FUNCTION_BLOCK PlixHandler
VAR_INPUT
	go :BOOL;

END_VAR
VAR_OUTPUT
	

END_VAR
VAR
	//Arduino				/////////////////////////////////////////
		//States
	Scanner					:USINT		:= 10;
	
		//Varibles
	WingUp					:USINT 		:=220;
	WingFlat				:USINT 		:=180;
	WingHDown				:USINT 		:=155;
	WingDown				:USINT 		:=80;
	WiggleDown				:USINT 		:=155;
	WiggleUP				:USINT 		:=190;
	FanHigh					:USINT 		:=115;
	FanLow					:USINT 		:=95;
	FanOff					:USINT 		:=89;
	FanReverse				:USINT 		:=74;
	WingGo					:USINT		:=20;
	FanGo					:USINT		:=30;

	//Stepper				/////////////////////////////////////////
	HaltStackStepper	: MC_Halt;
	EnableStackStepper	: MC_Power;
	MoveStackAbsolute	: MC_MoveAbsolute;
	ReadStackPosition	: MC_ReadActualPosition;
	SetStackPosition	: MC_SetPosition;
	StopStackStepper	: MC_Stop;
	ResetStackStepper	: MC_Reset;
	
		//Varibles
	StackStepperRun: BOOL;
	StackStepperPosition: LREAL;
	StackStepperVelocity: LREAL;
	StackStepperCurrentPosition: LREAL;
	StackStepperZeroPosition : BOOL;
	StackStepperStop: BOOL;
	StackStepperReset: BOOL;
	StackStepperHalt: BOOL;
	StackStepperHaltDone: BOOL;
	StackStepperAbsoluteDone: BOOL;
	StackStepperEnable: BOOL;
	
	Byte31IN: BYTE;
	StackSensor1: BOOL;
	Sensors: BYTE;
	StackSensor2: BOOL;
	StackSensor3: BOOL;
	Sensor4: BOOL;
	Sensor5: BOOL;
	PlixHandlerState: INT;
	BottomEndStop: BOOL;
	Boot: BOOL := TRUE;
	Calibrate 				:BOOL;
	NextState: INT;
	Single					:BOOL;
	Double					:BOOL;
	Zero					:BOOL;
	Start					:BOOL;
	//Stats					/////////////////////////////////////////
	Singles					:INT;
	Doubles					:INT;
	Zeros					:INT;
	Total					:INT;
	Wiggle					:INT;
	Count 					:INT		:= 0;
	Delay 					:TON;
	CycleTime				:REAL;
	EndTime					:REAL;
	AverageTime				:REAL;
	DoubleLoop: INT;
	Blast: BOOL;
	Cali: INT	 :=0;
	Velocity 				:LREAL :=800;
	ErrorID1		        : UDINT;
	
	Pig: BOOL;
END_VAR
VAR PERSISTENT				/////////////////////////////////////////
	
	//CutPoints				/////////////////////////////////////////
	PlixNumberScan			:INT;
	PlixNumberScanLeft		:INT;
	PlixNumberScanRight		:INT;
	NormalTopCut			:UINT;
	NormalBottomCut			:UINT;
	TopCut					:UINT;
	BottomCut				:UINT;
	DoubleTopCut			:UINT;
	DoubleBottomCut			:UINT;
	TopCutLeft				:INT;
	BottomCutLeft			:INT;
	TopCutRight				:INT;
	BottomCutRight			:INT;
	
	
	//Time					/////////////////////////////////////////

END_VAR

MoveStackAbsolute(
	Axis:= GVL.StackStepper, 
	Execute:= StackStepperRun, 
	Position:= StackStepperPosition, 
	Velocity:= StackStepperVelocity, 
	Acceleration:= 2518.53, 
	Deceleration:= 2518.53, 
	Jerk:= 10703.7,
	Done=> StackStepperAbsoluteDone, );
	
HaltStackStepper(
	Axis:= GVL.StackStepper, 
	Execute:= StackStepperHalt, 
	Deceleration:= 2518.53,  
	Done=> StackStepperHaltDone,
	ErrorID=> ErrorID1, );
	
EnableStackStepper(
	Axis:= GVL.StackStepper, 
	Enable:= StackStepperEnable, 
	Enable_Positive:= StackStepperEnable, 
	Enable_Negative:= StackStepperEnable, );

ReadStackPosition(
	Axis:= GVL.StackStepper, 
	Enable:= StackStepperEnable, 
	Position=> StackStepperCurrentPosition);	

SetStackPosition(
	Axis:= GVL.StackStepper, 
	Execute:= StackStepperZeroPosition, 
	Position:= 0, 
	Mode:= FALSE, 
	Options:= , 
	 );
	
StopStackStepper(
	Axis:= GVL.StackStepper, 
	Execute:= StackStepperStop, 
	Deceleration:= , 
	Jerk:= , 
	Options:= , 
	Done=> , 
	Busy=> , 
	Active=> , 
	CommandAborted=> , 
	Error=> , 
	ErrorID=> );
	
ResetStackStepper(
	Axis:= GVL.StackStepper, 
	Execute:= StackStepperReset, 
	Done=> , 
	Busy=> , 
	Error=> , 
	ErrorID=> );
	
	
	
	
	//Coms

IF go THEN
	StackStepperEnable := TRUE;
END_IF
StackSensor2 := GVL.Sensors2.0;
BottomEndStop :=GVL.Sensors2.1;
//StackStepperZeroPosition := TRUE;//sometimes after many restarts the position can be massive and cause problems 


CASE PlixHandlerState OF
	
	1:
		StackStepperZeroPosition := FALSE;
		StackStepperRun := FALSE;
		StackStepperHalt :=TRUE;
		IF StackStepperHaltDone THEN 
				PlixHandlerState :=NextState;
				StackStepperHalt :=FALSE;
		END_IF
		
	
	10:	
		IF Boot THEN
			StackStepperZeroPosition := TRUE;
			PlixHandlerState := 11;
		ELSE
			PlixHandlerState := 100;
		END_IF
		
	11://home bottom sensor
		StackStepperZeroPosition := FALSE;
		IF  BottomEndStop THEN//if not blocked drive down till blocked
			StackStepperPosition := -50000;
			StackStepperVelocity := 100;
			StackStepperRun := TRUE;
		ELSE 
			NextState :=20;
			PlixHandlerState :=1;
				
		END_IF
		
	20:
		IF  NOT BottomEndStop THEN//drive up till unblocked
			StackStepperPosition := 8000;
			StackStepperVelocity := 100;
			StackStepperRun := TRUE;
		ELSE 
			NextState :=30;
			PlixHandlerState :=1;	
		END_IF	
		
	30:
		Boot := FALSE;
		StackStepperZeroPosition := TRUE;//set position to zero just above endstop
		//StackStepperZeroPosition := FALSE;
		PlixHandlerState :=100;
	
	100:// home stack top
		StackStepperZeroPosition := FALSE;
		IF NOT StackSensor2 THEN//AND NOT StackSensor2 AND NOT StackSensor3 THEN
			StackStepperPosition := 200;
			StackStepperVelocity := Velocity;//make sure to change the amount of steps to plix pick up
			StackStepperRun := TRUE;
		ELSE 
			NextState :=200;
			PlixHandlerState :=1;
			
		END_IF
	200:
		StackStepperHalt :=FALSE;
		IF StackSensor2 THEN//AND  StackSensor2 AND  StackSensor3 THEN
			StackStepperPosition := 10000;
			StackStepperVelocity := Velocity;//make sure to change the amount of steps to plix pick up
			StackStepperRun := TRUE;
		ELSE 
			NextState :=300;
			PlixHandlerState :=1;
				
		END_IF
	300://fan on
		IF GVL.ArduinoBusyBit THEN//if  arduino is free then ask to change state
			GVL.FanDyno := FanHigh;
			GVL.ArduinoState := FanGo;
			PlixHandlerState :=400;
		END_IF
		
	400://up to head
		IF Blast THEN 
			GVL.StackBlast := TRUE;
		END_IF
		Blast := FALSE;
		StackStepperHalt :=FALSE;
		StackStepperPosition := StackStepperCurrentPosition + 50;
		StackStepperVelocity := Velocity;
		StackStepperRun := TRUE;
		PlixHandlerState :=500;
		
	500://down
		
		StackStepperRun := FALSE;
		IF StackStepperAbsoluteDone THEN
			GVL.StackBlast := FALSE;
		/////
			
			StackStepperPosition := StackStepperCurrentPosition - 400;
			StackStepperVelocity := Velocity;//make sure to change the amount of steps to plix pick up
			StackStepperRun := TRUE;
			StackStepperAbsoluteDone := FALSE;
			PlixHandlerState :=550;
			
		END_IF
		
	550:
		StackStepperRun := FALSE;
		IF StackStepperAbsoluteDone THEN
			NextState :=575;
			PlixHandlerState :=1;
				
		END_IF
		
	575:
		IF Calibrate THEN
			PlixHandlerState :=580;
		ELSE
			PlixHandlerState :=600;
		END_IF
		
	580:
		Delay(IN:=TRUE, PT:=T#1000MS);
      	IF Delay.Q THEN
        	Delay(IN:=FALSE);
			
			PlixHandlerState :=600;
		END_IF
	600://scan
		
		IF GVL.ArduinoBusyBit THEN//if arduino is free then ask to change state
			GVL.ArduinoState := Scanner;
			PlixHandlerState :=700;
		END_IF
	
	700:
		IF GVL.ArduinoBusyBit THEN//if arduino is free then ask to change state
			PlixHandlerState :=800;
		END_IF
	800://still hasnt written the new scan to beckhoff so we need to wait a little for it to loop on the arduino
	Delay(IN:=TRUE, PT:=T#500MS);
      	IF Delay.Q THEN
        	Delay(IN:=FALSE);
			
			PlixHandlerState :=900;
		END_IF
	900:
		IF NOT Calibrate THEN
			IF DoubleLoop > 0 THEN
				TopCut := DoubleTopCut;
				BottomCut := DoubleBottomCut;
				PlixHandlerState :=1000;
			ELSE
				TopCut := NormalTopCut;
				BottomCut := NormalBottomCut;
				PlixHandlerState :=1000;
			END_IF
		ELSE 
			PlixHandlerState :=1000;
		END_IF
	1000://decision
		IF GVL.Average > TopCut THEN
			Zero := TRUE;
			Blast := TRUE;
			PlixHandlerState :=2500;
		
		ELSIF  GVL.Average <= TopCut AND GVL.Average > BottomCut THEN
			Single := TRUE;
			PlixHandlerState :=2000;
			
		ELSIF GVL.Average <= BottomCut THEN
			
			Blast := TRUE;
			DoubleLoop := DoubleLoop +1;
			WiggleDown := WiggleDown - 25;
			WiggleUP := WiggleUP + 10;
			PlixHandlerState :=1025;
			
		END_IF
		IF Calibrate THEN
			IF Cali = 0 THEN
				Single := TRUE;
				NormalTopCut := GVL.Average + 100;
				NormalBottomCut := GVL.Average - 10;
				PlixHandlerState :=1025;
			ELSIF Cali = 1 THEN
				DoubleTopCut := GVL.Average + 100;
				DoubleBottomCut := GVL.Average - 20;
				PlixHandlerState :=2500;
			END_IF	
		END_IF
	//zero
		//blast stack
		//repick
	//double
		//wiggle
		//blast
		//rescan
	1025:
		IF DoubleLoop <= 1 THEN
			StackStepperPosition := StackStepperCurrentPosition - 150;
			StackStepperVelocity := Velocity;//make sure to change the amount of steps to plix pick up
			StackStepperRun := TRUE;
			PlixHandlerState :=1030;
		ELSE
			PlixHandlerState :=1050;
		END_IF
	1030:
		StackStepperRun := FALSE;
		
		IF StackStepperAbsoluteDone THEN
			Cali := 1;
			PlixHandlerState :=575;
		END_IF
	1050:
		
			IF DoubleLoop > 5 THEN
				Total := Total + 2;
				Double := TRUE;
				
				PlixHandlerState :=2000;
			ELSE
				PlixHandlerState :=1100;
			END_IF
		
	1100:
		Wiggle := Wiggle +1;
		IF GVL.ArduinoBusyBit THEN//if arduino is free then ask to change state
			GVL.WingSpeed := 60;
			GVL.FanDyno := WiggleDown;
			GVL.ArduinoState := WingGo;
			Delay(IN:=TRUE, PT:=T#500MS);
			IF Delay.Q THEN
				Delay(IN:=FALSE);
				GVL.DoubleJets := TRUE;
				//GVL.LeftAirJet := TRUE;
				PlixHandlerState := 1200; 
			END_IF
		END_IF
	1200:
		IF GVL.ArduinoBusyBit THEN//if arduino is free then ask to change state
			GVL.WingSpeed := 20;
			GVL.FanDyno := WiggleUP;
			GVL.ArduinoState := WingGo;
			Delay(IN:=TRUE, PT:=T#500MS);
			IF Delay.Q THEN
				Delay(IN:=FALSE);
				GVL.DoubleJets := FALSE;
				//GVL.RightAirJet := FALSE;
				PlixHandlerState := 1300;
			END_IF
		END_IF
	1300:
		IF GVL.ArduinoBusyBit THEN
			GVL.WingSpeed := 60;
			GVL.FanDyno :=WingFlat;
			GVL.ArduinoState := WingGo;
			
			Delay(IN:=TRUE, PT:=T#500MS);
			IF Delay.Q THEN
				Delay(IN:=FALSE);
				PlixHandlerState := 600;
			END_IF
		END_IF
	
	//////////////////////////////////////////////////
		
	2000:
		IF GVL.ArduinoBusyBit AND GVL.PlixRequest THEN //AND Pig THEN
			GVL.FanDyno := 74;
			Pig := FALSE;
			GVL.PlixRequest := FALSE;
			GVL.ArduinoState := FanGo;
			PlixHandlerState:=2200;
		END_IF
	2200:
			//GVL.FanDyno := 74;
			//GVL.ArduinoState := FanGo;
		Delay(IN:=TRUE, PT:=T#300MS);
		IF Delay.Q THEN
        	Delay(IN:=FALSE);
        	PlixHandlerState := 2300;
    	END_IF
	2300:
		IF GVL.ArduinoBusyBit THEN
			GVL.PlixShooter :=TRUE;
			GVL.PlixRequest := FALSE;
			PlixHandlerState := 2400;
		END_IF
	2400:
		Delay(IN:=TRUE, PT:=T#150MS);
		IF Delay.Q THEN
        	Delay(IN:=FALSE);
        	PlixHandlerState := 2500;
    	END_IF
	2500:
		IF GVL.ArduinoBusyBit THEN
			GVL.FanDyno := 89;
			GVL.ArduinoState := FanGo;
			PlixHandlerState := 2600;
		END_IF
	2600:
		Delay(IN:=TRUE, PT:=T#100MS);
		IF Delay.Q THEN
        	Delay(IN:=FALSE);
			GVL.PlixShooter :=FALSE;
        	PlixHandlerState := 2700;
    	END_IF
	2700:
		Delay(IN:=TRUE, PT:=T#2000MS);
		IF Delay.Q THEN
        	Delay(IN:=FALSE);
        	PlixHandlerState := 2800;
    	END_IF
	2800:
	//finishing up stats ant time and stuff
		PlixHandlerState :=100;
		DoubleLoop := 0;
		WiggleDown := 155;
		WiggleUP := 190;
		IF Single THEN
			Singles := Singles +1;
			Total := Total + 1;
		END_IF
		IF Double THEN
			Doubles := Doubles +1;
		END_IF
		Single := FALSE;
		Double := FALSE;
		EndTime := MAIN.TimeSeconds;	
		IF Singles > 1 THEN
			AverageTime := (EndTime - MAIN.GoTime)/Singles;
		END_IF
		
		CycleTime := EndTime - MAIN.StartTime;
		IF Calibrate THEN
			Singles := Singles -1;
			Blast := FALSE;
			Cali := 0;
			//TopCutLeft := GVL.AverageLeft - 40;
			//BottomCutLeft := AverageLeft - 66;
			//TopCutRight := AverageRight + 10;
			//BottomCutRight := AverageRight - 50;
			PlixHandlerState :=0;
			Calibrate := FALSE;
		END_IF
		
	
END_CASE

END_FUNCTION_BLOCK

(* stored: Version 1.1.0.1, ProductVersion 3.1.4024.2
   POU PlixHandler: Id {922d3b6a-8040-4ec2-a51e-3da1448b8660}, SpecialFunc None *)
